{attribute 'qualified_only'}
{attribute 'strict'}
TYPE E_PickPlaceStep :
(
	DO_NOTHING 	:= 0,
	MOVE_HAND 	:= 1,
	CHECK_GRIP	:= 2,
	USE_GRIP	:= 3
);
END_TYPE

(* stored: Version 1.1.0.1, ProductVersion 3.1.4024.9
   DUT E_PickPlaceStep: Id {52ec975c-0c83-41d0-952a-9b54d37767b8} *)
